//{attribute 'qualified_only'}
{attribute 'strict'}
TYPE eLM_State_Machine :
(
		LM_Off 			:= 0 ,
		LM_Init 		:= 1 ,
		LM_Ready 		:= 2 ,
		LM_CodeSend 	:= 3 ,
		LM_MarkCommand 	:= 4 ,
		LM_Feedback 	:= 5 
);
END_TYPE

(* stored: Version 1.1.0.1, ProductVersion 3.1.4024.3
   EnumerationTextList eLM_State_Machine: Id {5594767f-7fd9-4be5-a366-607e32dc8326} *)
